// TIA Portal V17 export
// export: Created 2026-05-13T14:55:42.0373285Z, ExportSetting WithDefaults, DisplayName Totally Integrated Automation Portal, DisplayVersion V17 Update 4, DisplayName TIA Portal Openness, DisplayVersion V17 Update 4, DisplayName TIA Portal Version Control Interface, DisplayVersion V17, DisplayName SINAMICS Startdrive Advanced, DisplayVersion V17, DisplayName SINAMICS Startdrive G130, G150, S120, S150, SINAMICS MV, S210, DisplayVersion V17, DisplayName SINAMICS Startdrive G110M, G120, G120C, G120D, G120P, G115D, DisplayVersion V17, DisplayName STEP 7 Professional, DisplayVersion V17 Update 4, DisplayName STEP 7 Safety, DisplayVersion V17, DisplayName WinCC Professional, DisplayVersion V17 Update 4
FUNCTION_BLOCK "HMI弹窗"   // FB1, SCL
{ S7_Optimized_Access := 'TRUE' }
VERSION : 0.1
// stored: AutoNumber true, IsIECCheckEnabled false, IsRetainMemResEnabled false, MemoryReserve 100, SetENOAutomatically false, UDAEnableTagReadback false
   VAR_INPUT
      DoubleClickTime : Time := T#800MS;
      CompID : Int;   // 部件唯一ID（>0）
   END_VAR
   VAR_IN_OUT
      Comp : "UDT_ComponentPopup";   // 单个部件
      Active : "UDT_ActivePopup";   // 全局激活区（共享）
   END_VAR
   VAR_TEMP
      R_Click : Bool;
      tNow : Time;
      tDiff : Time;
      i : Int;
   END_VAR
BEGIN
   // ========== 1. 上升沿检测 ==========
   #R_Click := #Comp.ClickTrig AND NOT #Comp.LastClick;
   #Comp.LastClick := #Comp.ClickTrig;

   #tNow := TIME_TCK();

   // ========== 2. 点击逻辑 ==========
   IF #R_Click THEN
       IF #Comp.ClickCount = 0 THEN
           // ===== 首次点击 → 打开弹窗，把部件数据复制到激活区 =====
           #Comp.ClickCount := 1;
           #Comp.FirstClickTime := #tNow;
           #Comp.Active := TRUE;

           #Active.ActiveID := #CompID;
           #Active.Visible := TRUE;
           #Active.Confirmed := FALSE;     // 清确认标志
           #Active.ConfirmBtn := FALSE;
           #Active.CancelBtn := FALSE;

           // 复制当前部件值 → 激活区（让HMI显示原值）
           FOR #i := 1 TO 8 DO
               #Active.Switch[#i] := #Comp.Switch[#i];
               #Active.RealValue[#i] := #Comp.RealValue[#i];
           END_FOR;
           #Active.InfoTitle := #Comp.InfoTitle;
           #Active.InfoMessage := #Comp.InfoMessage;
           #Active.InfoSpare1 := #Comp.InfoSpare1;
           #Active.InfoSpare2 := #Comp.InfoSpare2;

           // 设置可见性
           FOR #i := 1 TO 8 DO
               #Active.SwitchEnable[#i] := (#i <= #Comp.SwitchCnt);
               #Active.RealEnable[#i] := (#i <= #Comp.RealCnt);
           END_FOR;
           FOR #i := 1 TO 4 DO
               #Active.InfoEnable[#i] := (#i <= #Comp.InfoCnt);
           END_FOR;

       ELSE
           // ===== 双击窗口内再次点击 → 取消并隐藏（丢弃修改）=====
           #tDiff := #tNow - #Comp.FirstClickTime;
           IF #tDiff <= #DoubleClickTime THEN
               #Comp.Active := FALSE;
               #Comp.ClickCount := 0;
               #Active.Visible := FALSE;
               #Active.ActiveID := 0;
               FOR #i := 1 TO 8 DO
                   #Active.SwitchEnable[#i] := FALSE;
                   #Active.RealEnable[#i] := FALSE;
               END_FOR;
               FOR #i := 1 TO 4 DO
                   #Active.InfoEnable[#i] := FALSE;
               END_FOR;
               // ⚠ 不写回 Comp，丢弃HMI上的临时修改
           ELSE
               // 超时算新一轮首次点击
               #Comp.ClickCount := 1;
               #Comp.FirstClickTime := #tNow;
           END_IF;
       END_IF;
   END_IF;

   // ========== 3. 双击窗口超时清计数 ==========
   IF #Comp.ClickCount = 1 THEN
       IF (#tNow - #Comp.FirstClickTime) > #DoubleClickTime THEN
           #Comp.ClickCount := 0;
       END_IF;
   END_IF;

   // ========== 4. 当此部件激活时，处理确认/取消 ==========
   IF #Comp.Active AND (#Active.ActiveID = #CompID) THEN

       // ===== 确认按钮：把激活区的值提交到部件 =====
       IF #Active.ConfirmBtn THEN
           #Active.ConfirmBtn := FALSE;     // 自复位

           // ✅ 只在确认时写回部件
           FOR #i := 1 TO 8 DO
               #Comp.Switch[#i] := #Active.Switch[#i];
               #Comp.RealValue[#i] := #Active.RealValue[#i];
           END_FOR;

           #Active.Confirmed := TRUE;       // 给主程序判断用

           // 确认后关闭弹窗（按需保留/取消）
           #Active.Visible := FALSE;
           #Active.ActiveID := 0;
           #Comp.Active := FALSE;
           #Comp.ClickCount := 0;
           FOR #i := 1 TO 8 DO
               #Active.SwitchEnable[#i] := FALSE;
               #Active.RealEnable[#i] := FALSE;
           END_FOR;
           FOR #i := 1 TO 4 DO
               #Active.InfoEnable[#i] := FALSE;
           END_FOR;
       END_IF;

       // ===== 取消按钮：丢弃修改，关闭弹窗 =====
       IF #Active.CancelBtn THEN
           #Active.CancelBtn := FALSE;
           #Active.Visible := FALSE;
           #Active.ActiveID := 0;
           #Comp.Active := FALSE;
           #Comp.ClickCount := 0;
           FOR #i := 1 TO 8 DO
               #Active.SwitchEnable[#i] := FALSE;
               #Active.RealEnable[#i] := FALSE;
           END_FOR;
           FOR #i := 1 TO 4 DO
               #Active.InfoEnable[#i] := FALSE;
           END_FOR;
           // ⚠ 不写回 Comp
       END_IF;

   END_IF;
END_FUNCTION_BLOCK
